FUNCTION_BLOCK SifbIntLed
  (* Standard: 61499-2 *)
  (* Version 0.1, 2019-00-29, hpea485, UOA *)
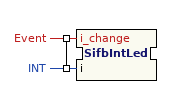
  EVENT_INPUT
    i_change WITH i;
  END_EVENT
  VAR_INPUT
    i : INT;
  END_VAR
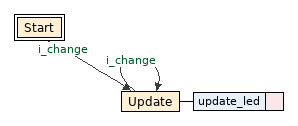
  EC_STATES
    Start;
    Update : update_led;
  END_STATES
  EC_TRANSITIONS
    Start TO Update := i_change;
    Update TO Update := i_change;
  END_TRANSITIONS
  ALGORITHM update_led IN C:
LED = me->i;
  END_ALGORITHM
END_FUNCTION_BLOCK
